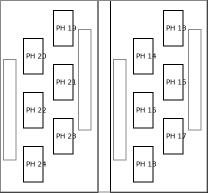
VISUALIZATION VISU_PhEnable_M3  // 208x193
    RoundedRectangle (0,0 98x193)
        toggle PRG_PRINT.sAdsPrintGroup[4].bI_Enable
    Rectangle (53,10 20x36), colour toggle: PRG_PRINT.sAdsPrintHead[19].bI_Enable
        toggle PRG_PRINT.sAdsPrintHead[19].bI_Enable
    Rectangle (23,38 20x36), colour toggle: PRG_PRINT.sAdsPrintHead[20].bI_Enable
        toggle PRG_PRINT.sAdsPrintHead[20].bI_Enable
    Rectangle (53,64 20x36), colour toggle: PRG_PRINT.sAdsPrintHead[21].bI_Enable
        toggle PRG_PRINT.sAdsPrintHead[21].bI_Enable
    Rectangle (23,92 20x36), colour toggle: PRG_PRINT.sAdsPrintHead[22].bI_Enable
        toggle PRG_PRINT.sAdsPrintHead[22].bI_Enable
    Rectangle (53,118 20x36), colour toggle: PRG_PRINT.sAdsPrintHead[23].bI_Enable
        toggle PRG_PRINT.sAdsPrintHead[23].bI_Enable
    Rectangle (23,146 20x36), colour toggle: PRG_PRINT.sAdsPrintHead[24].bI_Enable
        toggle PRG_PRINT.sAdsPrintHead[24].bI_Enable
    Rectangle (15,46 36x20), angle 270, "PH 20", colour toggle: PRG_PRINT.sAdsPrintHead[20].bI_Enable
    Rectangle (45,18 36x20), angle 270, "PH 19", colour toggle: PRG_PRINT.sAdsPrintHead[19].bI_Enable
    Rectangle (45,72 36x20), angle 270, "PH 21", colour toggle: PRG_PRINT.sAdsPrintHead[21].bI_Enable
    Rectangle (15,100 36x20), angle 270, "PH 22", colour toggle: PRG_PRINT.sAdsPrintHead[22].bI_Enable
    Rectangle (45,126 36x20), angle 270, "PH 23", colour toggle: PRG_PRINT.sAdsPrintHead[23].bI_Enable
    Rectangle (15,154 36x20), angle 270, "PH 24", colour toggle: PRG_PRINT.sAdsPrintHead[24].bI_Enable
    Frame (78,29 13x101)
        shows _VISU_PcMiniVertical(m_Inst := PRG_PRINT.FB_PC[7])
    Frame (3,59 13x101)
        shows _VISU_PcMiniVertical(m_Inst := PRG_PRINT.FB_PC[8])
    RoundedRectangle (110,0 98x193)
        toggle PRG_PRINT.sAdsPrintGroup[3].bI_Enable
    Rectangle (163,10 20x36), colour toggle: PRG_PRINT.sAdsPrintHead[13].bI_Enable
        toggle PRG_PRINT.sAdsPrintHead[13].bI_Enable
    Rectangle (133,38 20x36), colour toggle: PRG_PRINT.sAdsPrintHead[14].bI_Enable
        toggle PRG_PRINT.sAdsPrintHead[14].bI_Enable
    Rectangle (163,64 20x36), colour toggle: PRG_PRINT.sAdsPrintHead[15].bI_Enable
        toggle PRG_PRINT.sAdsPrintHead[15].bI_Enable
    Rectangle (133,92 20x36), colour toggle: PRG_PRINT.sAdsPrintHead[16].bI_Enable
        toggle PRG_PRINT.sAdsPrintHead[16].bI_Enable
    Rectangle (163,118 20x36), colour toggle: PRG_PRINT.sAdsPrintHead[17].bI_Enable
        toggle PRG_PRINT.sAdsPrintHead[17].bI_Enable
    Rectangle (133,146 20x36), colour toggle: PRG_PRINT.sAdsPrintHead[18].bI_Enable
        toggle PRG_PRINT.sAdsPrintHead[18].bI_Enable
    Rectangle (125,46 36x20), angle 270, "PH 14", colour toggle: PRG_PRINT.sAdsPrintHead[14].bI_Enable
    Rectangle (155,18 36x20), angle 270, "PH 13", colour toggle: PRG_PRINT.sAdsPrintHead[13].bI_Enable
    Rectangle (155,72 36x20), angle 270, "PH 15", colour toggle: PRG_PRINT.sAdsPrintHead[15].bI_Enable
    Rectangle (125,100 36x20), angle 270, "PH 16", colour toggle: PRG_PRINT.sAdsPrintHead[16].bI_Enable
    Rectangle (155,126 36x20), angle 270, "PH 17", colour toggle: PRG_PRINT.sAdsPrintHead[17].bI_Enable
    Rectangle (125,154 36x20), angle 270, "PH 18", colour toggle: PRG_PRINT.sAdsPrintHead[18].bI_Enable
    Frame (188,29 13x101)
        shows _VISU_PcMiniVertical(m_Inst := PRG_PRINT.FB_PC[5])
    Frame (113,59 13x101)
        shows _VISU_PcMiniVertical(m_Inst := PRG_PRINT.FB_PC[6])
END_VISUALIZATION

(* stored: Version 1.1.0.1, ProductVersion 3.1.4024.9
   Visu VISU_PhEnable_M3: Id {535cf4ec-4817-469a-9485-74b1ae587f18} *)
